(* PLC project Generated.project, CODESYS CODESYS V3.5 SP19 Patch 1 *)
(* stored: creationDateTime 2026-08-24T16:19:47.884736, modificationDateTime 2026-08-24T16:19:47.884736 *)

(* ======================================================================= ⚙️ ST_WinchSpeedConfig — Configuration des plages de vitesse linéaire ─────────────────────────────────────────────────────────────── 🎯 Rôle : Caractérisation des plages de vitesse mesurée par palier (m/s) 📄 Doc métier : DOC/AF/AF_Partie-10_Fonction_Winch_v2.0.md ======================================================================= *)
TYPE ST_WinchSpeedConfig : STRUCT
  MaxMeasuredSpeedMps : REAL;  (* Vitesse maximale mesuree de reference (m/s) *)
  SpeedBandMaxMps : ARRAY[1..5] OF REAL;  (* Plafonds vitesse mesuree par palier (m/s) *)
  SpeedBandHysteresisMps : REAL;  (* Hysteresis anti-battement classement vitesse (m/s) *)
END_STRUCT;
END_TYPE
